// TIA Portal V20 export
DATA_BLOCK "InstCallGeneral"   // DB25
// stored: InstanceOfName CallGeneral, InstanceOfType FB
"CallGeneral"
   // VAR
   //    statClockByteOld { ExternalWritable := 'False'} : Byte;
   //    instLAF_PowerOnOff { ExternalWritable := 'False'} : "LAF_PowerOnOff";
   //    instLAF_ClockGen { ExternalWritable := 'False'} : "LAF_ClockGenerator";
   //    instLSNTP_Server { ExternalWritable := 'False'} : "LSNTP_Server";
   //    instHmiManager { ExternalWritable := 'False'} : "LAF_HmiHeaderSingleUnitManager";
   // END_VAR
BEGIN
END_DATA_BLOCK
